//-----------------------------------------------------------------------------------------------------------------
//
//  HAUD 2026.03.21
//
//  - MAPPING : output 
//
//    - Status information to extern
//      - memcpy, to maintain data consistency
//      - instatiates control structures at compile
//      - use of compiler defines
//      - cyclic validation for matching sizes
//-----------------------------------------------------------------------------------------------------------------
PROGRAM MAPPING_out
VAR CONSTANT
//-----------------------------------------------------------------------------------------------------------------
//  - compiler defines check
//    - you find the compiler defines in the plc project properties under section Compile
//-----------------------------------------------------------------------------------------------------------------
{IF defined (MOVER_MAP)}
  {info 'XTS_TRANSPORT_LAYER: - MOVER_MAPPING active'}
  bBypassMappingMover       : BOOL  := FALSE;
  bMoverSelector            : BOOL  := FALSE;
{ELSE}
  // HAUD 2026 04 20
  // - selector is now configurable via compile
  {IF defined (MOVER_SELECTOR)}
    {info 'XTS_TRANSPORT_LAYER: - MOVER_SELECTOR active'}
    bBypassMappingMover     : BOOL  := FALSE;
    bMoverSelector          : BOOL  := TRUE;
  {ELSE}
    bBypassMappingMover     : BOOL  := TRUE;
    bMoverSelector          : BOOL  := FALSE;
  {END_IF}
{END_IF}
//-----------------------------------------------------------------------------------------------------------------
//-----------------------------------------------------------------------------------------------------------------
{IF defined (STATION_MAP)}
  {info 'XTS_TRANSPORT_LAYER: - STATION_MAPPING active'}
  bBypassMappingStation     : BOOL  := FALSE;
{ELSE}
  bBypassMappingStation     : BOOL  := TRUE;
{END_IF}
END_VAR
VAR
//-----------------------------------------------------------------------------------------------------------------
//-----------------------------------------------------------------------------------------------------------------
  sMappingCheck             : STRING;
//-----------------------------------------------------------------------------------------------------------------
//-----------------------------------------------------------------------------------------------------------------
{IF defined (MOVER_MAP)}
  MoverState                : U_MOVER_STATE;
  MoverInfo                 : U_MOVER_INFO;
{ELSE}
  // HAUD 2026 04 20
  // - selector is now configurable via compile
  {IF defined (MOVER_SELECTOR)}
    MoverState              : U_MOVER_SELECTOR_STATE;
    MoverInfo               : U_MOVER_INFO;
  {ELSE}
    MoverState              : BYTE;
    MoverInfo               : BYTE;
  {END_IF}
{END_IF}
//-----------------------------------------------------------------------------------------------------------------
//-----------------------------------------------------------------------------------------------------------------
{IF defined (STATION_MAP)}
  StationState              : U_XTS_STATION_STATE;
{ELSE}
  StationState              : BYTE;
{END_IF}
//-----------------------------------------------------------------------------------------------------------------
//-----------------------------------------------------------------------------------------------------------------
{IF (defined (STATION_MAP)) OR (defined (MOVER_MAP)) OR (defined(MOVER_SELECTOR))}
  {info 'XTS_TRANSPORT_LAYER: - TransportState'}
  TransportState            : U_XTS_TRANSPORT_STATE;
{ELSE}
  // TransportState            : BYTE;
  // explicit mapping for this specific example!!
  TransportState    : U_XTS_TRANSPORT_STATE;

  AppState          : U_APP_STATE;
  InstanceState     : U_INSTANCE_STATE;
  TicketListState   : U_TICKET_LIST_STATE;
  TicketListOutput  : U_TICKET_LIST_DATA_OUTPUT;
{END_IF}
//-----------------------------------------------------------------------------------------------------------------
//-----------------------------------------------------------------------------------------------------------------
  szMoverInfo,
  szMoverState              : ARRAY[1..2] OF UDINT;

  szStationState            : ARRAY[1..2] OF UDINT;

  szTransportState          : ARRAY[1..2] OF UDINT;

  pMoverState               : pvoid;
  pMoverInfo                : pvoid;
END_VAR

//--------------------------------------------------------------------------------------------
//  - datafield size check
//--------------------------------------------------------------------------------------------
IF NOT Check() THEN RETURN; END_IF
//--------------------------------------------------------------------------------------------
//--------------------------------------------------------------------------------------------
//--------------------------------------------------------------------------------------------
//           destination,               source,                             size
//--------------------------------------------------------------------------------------------
IF NOT bBypassMappingMover
THEN
  IF NOT bMoverSelector
  THEN
    pMoverState   := ADR(GVL_XTS.MoverState);
    pMoverInfo    := ADR(GVL_XTS.MoverInfo);
  ELSE
    pMoverState   := ADR(GVL_XTS.MoverSelectorState);
    pMoverInfo    := ADR(GVL_XTS.MoverInfo);
  END_IF

  memcpy(ADR(MoverState),           pMoverState,                    SIZEOF(MoverState));
  memcpy(ADR(MoverInfo) ,           pMoverInfo ,                    SIZEOF(MoverInfo));
END_IF
//--------------------------------------------------------------------------------------------
//--------------------------------------------------------------------------------------------
IF NOT bBypassMappingStation
THEN
  memcpy(ADR(StationState),         ADR(GVL_XTS.StationState),       SIZEOF(StationState));
END_IF
//--------------------------------------------------------------------------------------------
//--------------------------------------------------------------------------------------------
//       destination,           source,                                    size
//-----------------------------------------------------------------------------------------
  memcpy(ADR(TransportState),   ADR(GVL_XTS.XtsTransportState),            SIZEOF(TransportState));
  memcpy(ADR(AppState),         ADR(GVL_APPLICATION.AppState),             SIZEOF(AppState));
  memcpy(ADR(InstanceState),    ADR(GVL_APPLICATION.InstanceState),        SIZEOF(InstanceState));
  memcpy(ADR(TicketListState),  ADR(GVL_APPLICATION.TicketListState),      SIZEOF(TicketListState));
  memcpy(ADR(TicketListOutput), ADR(GVL_APPLICATION.TicketListDataOutput), SIZEOF(TicketListOutput));
//-----------------------------------------------------------------------------------------
//-----------------------------------------------------------------------------------------
(*
IF NOT bBypassMappingStation OR
   NOT bBypassMappingMover
THEN
  memcpy(ADR(TransportState),       ADR(GVL_XTS.XtsTransportState),  SIZEOF(TransportState));
END_IF
*)
//--------------------------------------------------------------------------------------------
//--------------------------------------------------------------------------------------------
//           destination,               source,                             size
//--------------------------------------------------------------------------------------------
//-----------------------------------------------------------------------------------------

METHOD Check : BOOL
VAR_INPUT
END_VAR
//--------------------------------------------------------------------------------------------
// - check first if compiler defines were set
// - you'll find the compiler defines in the plc project properties
//--------------------------------------------------------------------------------------------
(*  HAUD - for this example the instances are controlling the XTS, they are hardwired in this programm
IF bBypassMappingMover AND
   bBypassMappingStation
THEN
  sMappingCheck         := 'NO_MAPPING_ACTIVE';
  RETURN;
END_IF
*)
//--------------------------------------------------------------------------------------------
// - check datafields for matching sizes
// - if you keep the unions true, this method is always true
//--------------------------------------------------------------------------------------------
IF NOT bMoverSelector
THEN
  szMoverState  [1]   := SIZEOF(MoverState);
  szMoverState  [2]   := SIZEOF(GVL_XTS.MoverState);
ELSE
  szMoverState  [1]   := SIZEOF(MoverState);
  szMoverState  [2]   := SIZEOF(GVL_XTS.MoverSelectorState);
END_IF
szMoverInfo     [1]   := SIZEOF(MoverInfo);
szMoverInfo     [2]   := SIZEOF(GVL_XTS.MoverInfo);

IF NOT (bBypassMappingMover)
THEN
  IF NOT (szMoverState[1] = szMoverState[2])
  THEN
    sMappingCheck       := 'MoverState CHECK_ERROR';
    RETURN;
  END_IF

  IF NOT (szMoverInfo[1] = szMoverInfo[2])
  THEN
    sMappingCheck       := 'MoverInfo CHECK_ERROR';
    RETURN;
  END_IF
END_IF
//--------------------------------------------------------------------------------------------
//--------------------------------------------------------------------------------------------
szStationState  [1]   := SIZEOF(StationState);
szStationState  [2]   := SIZEOF(GVL_XTS.StationState);

IF NOT (bBypassMappingStation)
THEN
  IF NOT (szStationState[1] = szStationState[2])
  THEN
    sMappingCheck       := 'StationState CHECK_ERROR';
    RETURN;
  END_IF
END_IF
//--------------------------------------------------------------------------------------------
//--------------------------------------------------------------------------------------------
szTransportState[1]   := SIZEOF(TransportState);
szTransportState[2]   := SIZEOF(GVL_XTS.XtsTransportState);

IF NOT (bBypassMappingStation) OR
   NOT (bBypassMappingMover)
THEN
  IF NOT (szTransportState[1] = szTransportState[2])
  THEN
    sMappingCheck       := 'TransportState CHECK_ERROR';
    RETURN;
  END_IF
END_IF
//--------------------------------------------------------------------------------------------
//--------------------------------------------------------------------------------------------
//--------------------------------------------------------------------------------------------
//--------------------------------------------------------------------------------------------
sMappingCheck           := 'CHECK_DONE';
Check                   := TRUE;
//--------------------------------------------------------------------------------------------
//--------------------------------------------------------------------------------------------
END_METHOD

END_PROGRAM

(* stored: Version 1.1.0.1, ProductVersion 3.1.4026.18
   POU MAPPING_out: Id {b57f8ea9-4be8-44e1-a8de-2edb8d80a71f}, SpecialFunc None
   Method Check: Id {e2b027a8-a8c1-4ce6-b28e-ef5596bae8e6} *)
